// TIA Portal V16 export
// export: Created 2021-08-10T09:05:00.1501274Z, ExportSetting WithDefaults, WithReadOnly, DisplayName Totally Integrated Automation Portal, DisplayVersion V16, DisplayName TIA Portal Version Control Interface, DisplayVersion V16, DisplayName TIA Portal Openness, DisplayVersion V16, DisplayName TIA Portal Teamcenter Gateway, DisplayVersion V16, DisplayName SINAMICS Startdrive Advanced, DisplayVersion V16, DisplayName SINAMICS Startdrive G130, G150, S120, S150, SINAMICS MV, S210, DisplayVersion V16, DisplayName SINAMICS Startdrive G110M, G120, G120C, G120D, G120P, DisplayVersion V16, DisplayName STEP 7 Professional, DisplayVersion V16, DisplayName STEP 7 Safety, DisplayVersion V16, DisplayName WinCC Unified SCADA Engineering System, DisplayVersion V16
FUNCTION "fcSetHMIStatusSimulation" : Void   // FC333, FBD
TITLE = Sets HMI Status
{ S7_Optimized_Access := 'TRUE' }
VERSION : 0.1
// Wrapper function for setting the HMI status of a device
// 
// In order of priority:
// 1. E-stop
// 2. Error
// 3. Forward/Work Position
// 4. Reverse/Home Position
// 5. Forward/Work On
// 6. Reverse/Home On
// 7. None
// stored: AutoNumber true, CodeModifiedDate 2020-08-01T14:00:45.2523905Z, CompileDate 2021-07-03T08:38:37.6631079Z, CreationDate 2020-02-26T07:34:28.9567791Z, HandleErrorsWithinBlock false, InterfaceModifiedDate 2019-07-16T09:38:07.8023625Z, IsConsistent true, IsIECCheckEnabled false, IsKnowHowProtected false, IsWriteProtected false, LibraryConformanceStatus Warning: The object contains access to global PLC constants., LibraryType fcSetHMIStatusSimulation V 3.0.4, LibraryTypeVersionGuid 66f3681c-ca78-4b7d-9ef9-bd50d3b993d6, ModifiedDate 2020-08-01T14:00:53.126388Z, ParameterModified 2019-07-16T09:38:07.8023625Z, PLCSimAdvancedSupport true, SetENOAutomatically false, StructureModified 2019-07-16T09:38:07.8023625Z, UDAEnableTagReadback false
   VAR_INPUT
      bInEstop : Bool;
      bInError : Bool;
      bInForwardWork : Bool;
      bInReverseHome : Bool;
      bInOnForwardWork : Bool;
      bInOnReverseHome : Bool;
      bInSimulate : Bool;
   END_VAR
   VAR_OUTPUT
      iOutStatus : Int;
   END_VAR
BEGIN

REGION Network 1: Set Reverse/Home On
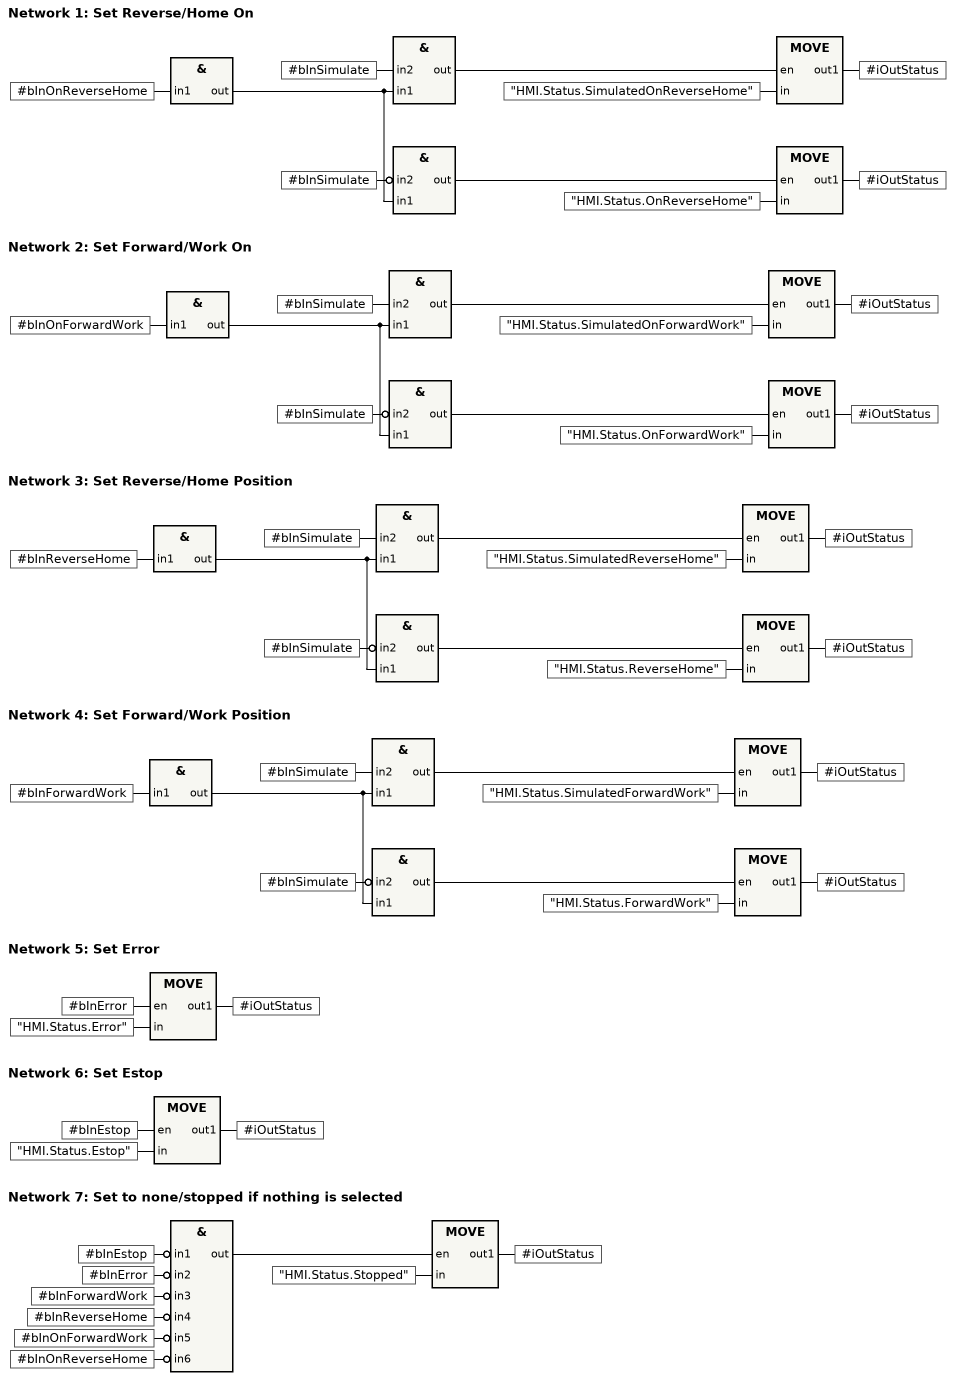
   IF #bInSimulate AND #bInOnReverseHome THEN #iOutStatus := "HMI.Status.SimulatedOnReverseHome"; END_IF;
   IF NOT #bInSimulate AND #bInOnReverseHome THEN #iOutStatus := "HMI.Status.OnReverseHome"; END_IF;
END_REGION

REGION Network 2: Set Forward/Work On
   IF #bInSimulate AND #bInOnForwardWork THEN #iOutStatus := "HMI.Status.SimulatedOnForwardWork"; END_IF;
   IF NOT #bInSimulate AND #bInOnForwardWork THEN #iOutStatus := "HMI.Status.OnForwardWork"; END_IF;
END_REGION

REGION Network 3: Set Reverse/Home Position
   IF #bInSimulate AND #bInReverseHome THEN #iOutStatus := "HMI.Status.SimulatedReverseHome"; END_IF;
   IF NOT #bInSimulate AND #bInReverseHome THEN #iOutStatus := "HMI.Status.ReverseHome"; END_IF;
END_REGION

REGION Network 4: Set Forward/Work Position
   IF #bInSimulate AND #bInForwardWork THEN #iOutStatus := "HMI.Status.SimulatedForwardWork"; END_IF;
   IF NOT #bInSimulate AND #bInForwardWork THEN #iOutStatus := "HMI.Status.ForwardWork"; END_IF;
END_REGION

REGION Network 5: Set Error
   IF #bInError THEN #iOutStatus := "HMI.Status.Error"; END_IF;
END_REGION

REGION Network 6: Set Estop
   IF #bInEstop THEN #iOutStatus := "HMI.Status.Estop"; END_IF;
END_REGION

REGION Network 7: Set to none/stopped if nothing is selected
   IF NOT #bInEstop AND NOT #bInError AND NOT #bInForwardWork AND NOT #bInReverseHome AND NOT #bInOnForwardWork AND NOT #bInOnReverseHome THEN
       #iOutStatus := "HMI.Status.Stopped";
   END_IF;
END_REGION

REGION Network 8: Set ENO
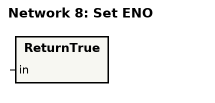
   ENO := TRUE;
   RETURN;
END_REGION
END_FUNCTION
